FUNCTION_BLOCK INTERNAL LCA_CAL
VAR_INPUT
	PSratedV 		: REAL; //kV
	RequiredChargeV	: REAL; //kV
	LoadCapacitance : REAL; //uF
	NumOfCharger	: INT := 1;
	wLCA			: BOOL;
END_VAR
VAR_OUTPUT
	TimeToChargeLoad 	 : REAL;
	RespectedPower		 : REAL;
END_VAR
VAR
	TotalPeakPowerRating : REAL := 9; //kJ/s
	TotalPeakChargeCurrent : REAL;
	AveChargeCurrent 	 : REAL; //A
	LoadStoredEnergy	 : REAL; //J
	Voltage				 : REAL; //
	Volt				 : ARRAY [0..480] OF REAL;
	t					 : ARRAY [0..480] OF REAL;
	deltaT				 : REAL; 
	Icharge				 : ARRAY [0..480] OF REAL;
	Power				 : ARRAY [0..480] OF REAL;
	i : INT := 1;
	j : INT := 1;
	
END_VAR

Volt[0] := 0;
t[0] := 0;
TotalPeakPowerRating := 9 * NumOfCharger;

IF wLCA = FALSE THEN 
	AveChargeCurrent := TotalPeakPowerRating / PSratedV;
	LoadStoredEnergy := 0.5*LoadCapacitance*LREAL_TO_REAL(EXPT(PSratedV, 2));
	//=+(D15*D7/D22)/350
	deltaT := (LoadCapacitance * PSratedV / AveChargeCurrent) / 350; //time step
	//=IF(C35>=(D$9*1000),0,D$22)
	//=+C33+B33*(D$26/1000)/(D$15*0.000001)
	IF Volt[0] >= (RequiredChargeV*1000.5) THEN 
		Icharge[0] := 0;
	ELSE
		Icharge[0] := AveChargeCurrent;
	END_IF
	
	FOR i := 1 TO 480 BY 1 DO 
			
		IF Volt[i] >= (RequiredChargeV*1000.5) THEN 
			Icharge[i] := 0;
		ELSE	
			Icharge[i] := AveChargeCurrent;
		END_IF
		Power[i] := Icharge[i]*Volt[i];
		t[i] := t[i-1]+ deltaT/1000;
		IF Volt[i] >= RequiredChargeV*1000*(0.98) AND Volt[i] <= RequiredChargeV*1000*(1.03) AND Power[i] <> 0 AND Power[i+1] = 0 THEN 
			TimeToChargeLoad := t[i];
			RespectedPower := Power[i];
		END_IF
		Volt[i] := Volt[i-1]+Icharge[i-1]*(deltaT/1000)/(LoadCapacitance*0.000001);
	END_FOR
ELSE//with LCA
	LoadStoredEnergy := 0.5*LoadCapacitance*0.000001*LREAL_TO_REAL(EXPT((RequiredChargeV*1000), 2));
	TotalPeakChargeCurrent := TotalPeakPowerRating*2/PSratedV;
	//IF(C36>=(D$9*1000),0,+IF(C36<500*D$7,D$24,D$24*(0.5+(D$7*1000-C36)/(D$7*1000))))
	deltaT := (LoadCapacitance*PSratedV/TotalPeakChargeCurrent)/350;
				
	IF Volt[i] >= (RequiredChargeV*1000) THEN 
		Icharge[0] := 0;
	ELSIF Volt[i] < (500*PSratedV) THEN
		Icharge[0] := TotalPeakChargeCurrent;
	ELSE
		Icharge[0] := TotalPeakChargeCurrent*(0.5+(PSratedV*1000-Volt[0])/(PSratedV*1000));
	END_IF
	
	FOR i := 1 TO 480 BY 1 DO
			
		IF Volt[i] >= (RequiredChargeV*1000) THEN 
			Icharge[i] := 0;
		ELSE
			IF Volt[i] < (500*PSratedV) THEN
				Icharge[i] := TotalPeakChargeCurrent;
			ELSE
				Icharge[i] := TotalPeakChargeCurrent*(0.5+(PSratedV*1000-Volt[i])/(PSratedV*1000));
			END_IF	
		END_IF
		Volt[i] := Volt[i-1]+Icharge[i-1]*(deltaT/1000)/(LoadCapacitance*0.000001);
		Power[i] := Icharge[i]*Volt[i];
		t[i] := t[i-1]+ deltaT/1000;
		IF Volt[i] >= RequiredChargeV*1000*(0.98) AND Volt[i] <= RequiredChargeV*1000*(1.03) AND Power[i] <> 0 AND Power[i+1] = 0 THEN 
			TimeToChargeLoad := t[i];
			RespectedPower := Power[i];
		END_IF
	END_FOR
END_IF;


IF i > 480 THEN
	i := 1;
END_IF

END_FUNCTION_BLOCK

(* stored: Version 1.1.0.1, ProductVersion 3.1.4024.11
   POU LCA_CAL: Id {a771c93a-8dfa-442a-b59f-33fb1819e105}, SpecialFunc None *)
